PROGRAM OK_Rep_Pupitre
VAR
	Voie_IOLink	 :BOOL;

	Rep_Pupitre				:FB_Rep_Ethercat_MURR;

	Joystick_Pupitre: FB_IOLink_MURR_MVP12;
END_VAR

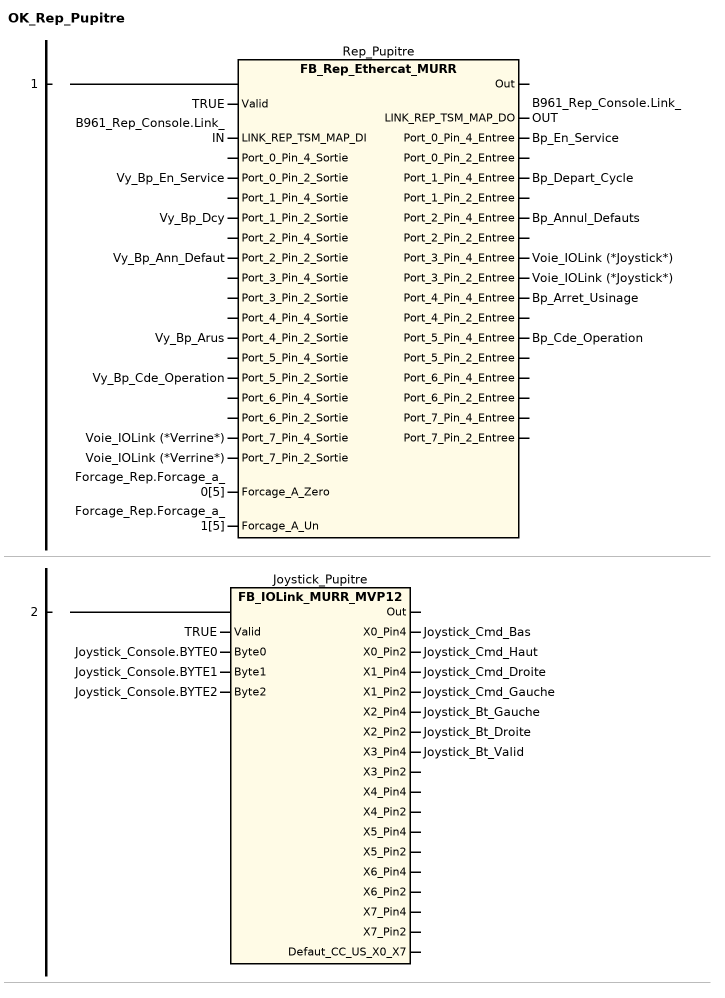
// NETWORK 1
Rep_Pupitre(
    Valid := TRUE,
    LINK_REP_TSM_MAP_DI := B961_Rep_Console.Link_IN,
    Port_0_Pin_2_Sortie := Vy_Bp_En_Service,
    Port_1_Pin_2_Sortie := Vy_Bp_Dcy,
    Port_2_Pin_2_Sortie := Vy_Bp_Ann_Defaut,
    Port_4_Pin_2_Sortie := Vy_Bp_Arus,
    Port_5_Pin_2_Sortie := Vy_Bp_Cde_Operation,
    Port_7_Pin_4_Sortie := Voie_IOLink (*Verrine*),
    Port_7_Pin_2_Sortie := Voie_IOLink (*Verrine*),
    Forcage_A_Zero := Forcage_Rep.Forcage_a_0[5],
    Forcage_A_Un := Forcage_Rep.Forcage_a_1[5],
    LINK_REP_TSM_MAP_DO => B961_Rep_Console.Link_OUT,
    Port_0_Pin_4_Entree => Bp_En_Service,
    Port_1_Pin_4_Entree => Bp_Depart_Cycle,
    Port_2_Pin_4_Entree => Bp_Annul_Defauts,
    Port_3_Pin_4_Entree => Voie_IOLink (*Joystick*),
    Port_3_Pin_2_Entree => Voie_IOLink (*Joystick*),
    Port_4_Pin_4_Entree => Bp_Arret_Usinage,
    Port_5_Pin_4_Entree => Bp_Cde_Operation); // FB_Rep_Ethercat_MURR

// NETWORK 2
Joystick_Pupitre(
    Valid := TRUE,
    Byte0 := Joystick_Console.BYTE0,
    Byte1 := Joystick_Console.BYTE1,
    Byte2 := Joystick_Console.BYTE2,
    X0_Pin4 => Joystick_Cmd_Bas,
    X0_Pin2 => Joystick_Cmd_Haut,
    X1_Pin4 => Joystick_Cmd_Droite,
    X1_Pin2 => Joystick_Cmd_Gauche,
    X2_Pin4 => Joystick_Bt_Gauche,
    X2_Pin2 => Joystick_Bt_Droite,
    X3_Pin4 => Joystick_Bt_Valid); // FB_IOLink_MURR_MVP12

END_PROGRAM

(* stored: Version 1.1.0.1
   POU OK_Rep_Pupitre: Id {7a67c669-f14e-4053-be2a-13d80eaf1e0e}, SpecialFunc None *)
